PROGRAM MAIN
VAR
	// Lakeshore 224 (Ethernet TCP Realtime interface)
	{attribute 'OPC.UA.DA' := '1'}
	LS224_TCP_RT:	FB_LAKESHORE_TCP_RT;	// LakeShore based on FB_TCP_RT_CLIENT

	// Lakeshore 336 (Ethernet TCP Realtime interface)
	{attribute 'OPC.UA.DA' := '1'}
	LS336_TCP_RT:	FB_LAKESHORE_TCP_RT;	// LakeShore based on FB_TCP_RT_CLIENT
	
	bDymmy	AT %I*:	BOOL;

END_VAR

		
LS224_TCP_RT(	in_sName			:= 'LS224_TCP_RT',
				in_nModel			:= 224,
				in_sCmdSuffix		:= '$0D$0A',
				in_sDeviceTcpIpAdr	:= '192.168.0.12',
				in_nDeviceTcpPort	:= 7777,
				in_nPeriod			:= 1200); 
		
LS336_TCP_RT(	in_sName			:= 'LS336_TCP_RT',
				in_nModel			:= 336,
				in_sCmdSuffix		:= '$0A',
				in_sDeviceTcpIpAdr	:= '192.168.0.80',
				in_nDeviceTcpPort	:= 7777,
				in_nPeriod			:= 1000);

END_PROGRAM

(* stored: Version 1.1.0.1, ProductVersion 3.1.4022.16
   POU MAIN: Id {4cb59fba-07cc-4017-b1f3-d17678eefef2}, SpecialFunc None *)
